// TIA Portal V17 export
// export: Created 2024-09-02T12:50:40.0906687Z, ExportSetting WithDefaults, DisplayName Totally Integrated Automation Portal, DisplayVersion V17, DisplayName TIA Portal Openness, DisplayVersion V17, DisplayName TIA Portal Version Control Interface, DisplayVersion V17, DisplayName STEP 7 Professional, DisplayVersion V17, DisplayName STEP 7 Safety, DisplayVersion V17, DisplayName WinCC Professional, DisplayVersion V17
TYPE "Scania_typ_Status"
// stored: IsFailsafeCompliant false
   STRUCT
      Res : Bool;
      Finished : Bool;
      "Finished OK" : Bool;
      "Finished NOK" : Bool;
      Bypass : Bool;
      Repaired : Bool;
      "OK Operator" : Bool;
      "NOK Operator" : Bool;
   END_STRUCT;
END_TYPE
